// Mitsubishi GX Works2 project: pneumatic_control_3   PLC: Q03UDV

PROGRAM MAIN
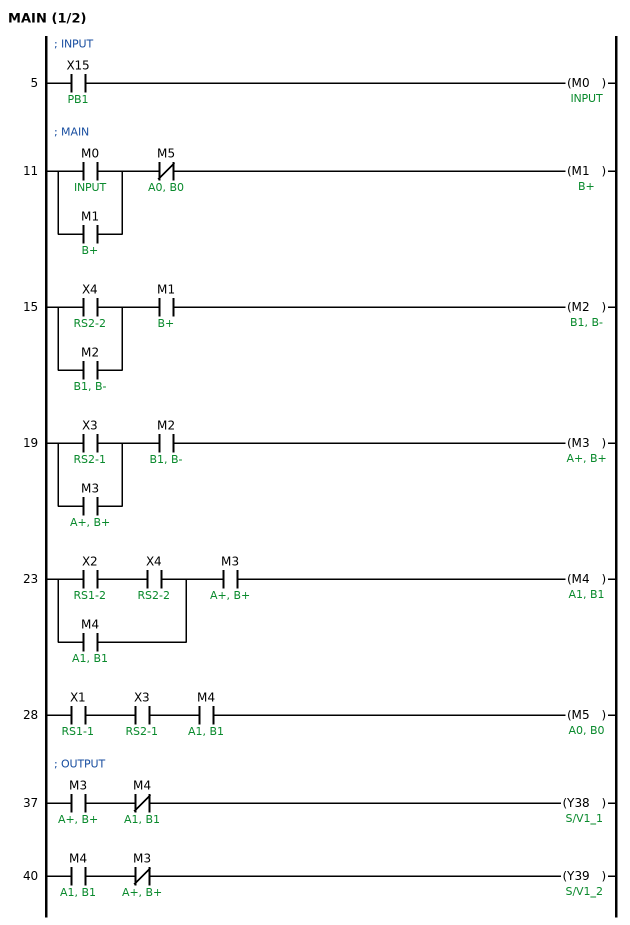
; INPUT
5     LD      X15  ; PB1
      OUT     M0  ; INPUT
; MAIN
11    LD      M0  ; INPUT
      OR      M1  ; B+
      ANI     M5  ; A0, B0
      OUT     M1  ; B+
15    LD      X4  ; RS2-2
      OR      M2  ; B1, B-
      AND     M1  ; B+
      OUT     M2  ; B1, B-
19    LD      X3  ; RS2-1
      OR      M3  ; A+, B+
      AND     M2  ; B1, B-
      OUT     M3  ; A+, B+
23    LD      X2  ; RS1-2
      AND     X4  ; RS2-2
      OR      M4  ; A1, B1
      AND     M3  ; A+, B+
      OUT     M4  ; A1, B1
28    LD      X1  ; RS1-1
      AND     X3  ; RS2-1
      AND     M4  ; A1, B1
      OUT     M5  ; A0, B0
; OUTPUT
37    LD      M3  ; A+, B+
      ANI     M4  ; A1, B1
      OUT     Y38  ; S/V1_1
40    LD      M4  ; A1, B1
      ANI     M3  ; A+, B+
      OUT     Y39  ; S/V1_2
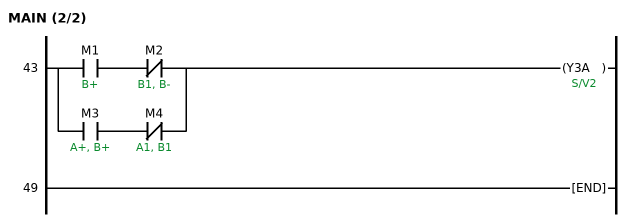
43    LD      M1  ; B+
      ANI     M2  ; B1, B-
      LD      M3  ; A+, B+
      ANI     M4  ; A1, B1
      ORB
      OUT     Y3A  ; S/V2
49    END
END_PROGRAM
